FUNCTION CheckBounds : DINT
VAR_INPUT
        index, lower, upper : DINT;
END_VAR
VAR
END_VAR

IF index<lower THEN
        CheckBounds := lower;
ELSIF index>upper THEN
        CheckBounds := upper;
ELSE
        CheckBounds := index;
END_IF

END_FUNCTION

(* stored: Version 1.1.0.1, ProductVersion 3.1.0.25
   POU CheckBounds: Id {cee9da00-acfc-4f83-a07a-0160f34b636f} *)
